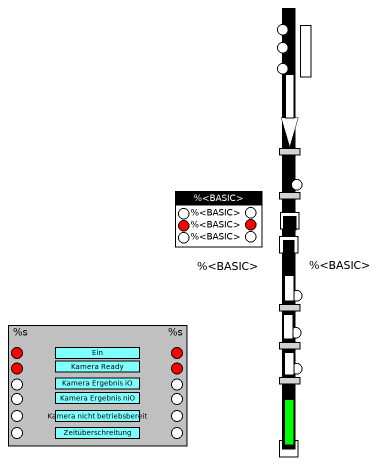
[picture p229: ZUFUEHRUNG_160POL (HMI screen)]
ellipse at (269,34)-(280,45): alarm colour if ST03_421_B63_5.BitInToCheck; tooltip ST03_421_B63_5
embedded screen at (273,66)-(290,139): SIGNS_ARROWDOWN
rounded rectangle at (272,204)-(291,221): alarm colour if ST03_422_B64_0.BitInToCheck; tooltip ST03_422_B64_0
ellipse at (269,55)-(280,66): alarm colour if ST03_421_B63_6.BitInToCheck; tooltip ST03_421_B63_6
ellipse at (269,16)-(280,27): alarm colour if ST03_421_B63_4.BitInToCheck; tooltip ST03_421_B63_4
ellipse at (283,282)-(294,293): alarm colour if ST03_422_B64_3.BitInToCheck; tooltip ST03_422_B64_3
rounded rectangle at (271,432)-(290,449): alarm colour if ST03_422_B64_4.BitInToCheck; tooltip ST03_422_B64_4
embedded screen at (0,317)-(179,437): ZLIB_SENSOPART_2
rectangle at (276,266)-(286,291): invisible if ST03_160pol_Zufuehrung.CamResult < 11; alarm colour if ST03_160pol_Zufuehrung.CamResult = 99
rectangle at (276,267)-(286,293): invisible if ST03_160pol_Zufuehrung.CamResult >= 11 OR NOT ST03_422_B64_3.BitInToCheck
rectangle at (276,391)-(286,437): invisible if NOT ST03_422_B64_4.BitInToCheck; alarm colour if ST03_Main.Result=RESULT_NOK
rectangle at (271,296)-(292,303): alarm colour if ST03_422_B64_1.ValveSensor; tooltip ST03_422_B64_1
rectangle at (271,184)-(292,191): alarm colour if ST03_421_B63_2.ValveSensor; tooltip ST03_421_B63_2
rectangle at (271,140)-(292,147): alarm colour if ST03_421_B63_0.ValveSensor; tooltip ST03_421_B63_0
rectangle at (275,212)-(286,226): alarm colour if ST03_421_B63_7.BitInToCheck
ellipse at (283,171)-(294,182): alarm colour if ST03_421_B63_7.BitInToCheck; tooltip ST03_421_B63_7
rounded rectangle at (292,17)-(303,69): alarm colour if ST03_Init_Lockings.b_freiFuerSG; tooltip b_freiFuerSG
embedded screen at (0,317)-(179,438): ZLIB_SENSOPART_6
ellipse at (282,319)-(293,330): alarm colour if ST03_423_B65_2.BitInToCheck; tooltip ST03_423_B65_2
rectangle at (275,305)-(285,330): invisible if ST03_160pol_Zufuehrung.CamResult2 < 11; alarm colour if ST03_160pol_Zufuehrung.CamResult2 = 99
rectangle at (275,306)-(285,331): invisible if ST03_160pol_Zufuehrung.CamResult2 >= 11 OR NOT ST03_423_B65_2.BitInToCheck
rectangle at (271,334)-(292,341): alarm colour if ST03_423_B65_0.ValveSensor; tooltip ST03_423_B65_0
ellipse at (283,355)-(294,366): alarm colour if ST03_423_B65_5.BitInToCheck; tooltip ST03_423_B65_5
rectangle at (276,343)-(286,365): invisible if ST03_160pol_Zufuehrung.CamResult3 < 11; alarm colour if ST03_160pol_Zufuehrung.CamResult3 = 99
rectangle at (276,344)-(286,367): invisible if ST03_160pol_Zufuehrung.CamResult3 >= 11 OR NOT ST03_423_B65_5.BitInToCheck
rectangle at (271,369)-(292,376): alarm colour if ST03_423_B65_4.ValveSensor; tooltip ST03_423_B65_4
rectangle at (299,245)-(374,270): text "%<BASIC>"; shows 'NIO Kamera'
rectangle at (187,246)-(265,271): text "%<BASIC>"; shows 'NIO Kamera'
rounded rectangle at (271,228)-(290,245): alarm colour if ST03_423_B66_0.BitInToCheck; tooltip ST03_423_B66_0
rectangle at (275,232)-(286,246): alarm colour if ST03_421_B63_7.BitInToCheck
rectangle at (167,196)-(254,239): shows 'Tank voll'
rectangle at (182,195)-(233,214): text "%<BASIC>"; shows 'bereit'
ellipse at (237,199)-(248,210): alarm colour if ST03_70U3_1.BitInToCheck
ellipse at (170,200)-(181,211): alarm colour if ST03_71U3_1.BitInToCheck
rectangle at (182,207)-(233,226): text "%<BASIC>"; shows 'Störung'
ellipse at (237,211)-(248,222): invisible if MP.ST03.SGM_3621; alarm colour if ST03_70U3_2.BitInToCheck
ellipse at (170,212)-(181,223): invisible if MP.ST03.SGM_3621; alarm colour if ST03_71U3_2.BitInToCheck
rectangle at (182,219)-(233,238): text "%<BASIC>"; shows 'Störung'
ellipse at (237,223)-(248,234): alarm colour if ST03_70U3_3.BitInToCheck
ellipse at (170,224)-(181,235): alarm colour if ST03_71U3_3.BitInToCheck
rectangle at (167,183)-(254,197): text "%<BASIC>"; shows 'li_Drucker_re'
3 more shapes without text or variables
6 elements of other kinds (tables, trends, ...) not read
*)

(* Visualisation zLibrary/ept/Zuführungen/ZUFUEHRUNG_191POL
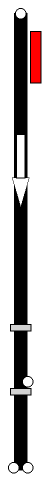
embedded screen at (9,126)-(26,199): SIGNS_ARROWDOWN
ellipse at (12,0)-(23,11): alarm colour if ST03_541_B69_0.BitInToCheck; tooltip ST03_541_B69_0
ellipse at (19,368)-(30,379): alarm colour if ST03_541_B69_6.BitInToCheck; tooltip ST03_541_B69_6
rectangle at (7,380)-(28,387): alarm colour if ST03_541_B69_4.ValveSensor; tooltip ST03_541_B69_3
rectangle at (7,316)-(28,323): alarm colour if ST03_541_B69_2.ValveSensor; tooltip ST03_541_B69_1
rounded rectangle at (27,23)-(38,75): alarm colour if ST03_Init_Lockings.b_freiFuerSG; tooltip b_freiFuerSG
ellipse at (19,454)-(30,465): alarm colour if ST03_542_B70_0.BitInToCheck; tooltip ST03_542_B70_0
ellipse at (5,454)-(16,465): alarm colour if ST03_541_B69_7.BitInToCheck; tooltip ST03_542_B70_0
2 more shapes without text or variables
*)

(* Visualisation zLibrary/ept/Zuführungen/ZUFUEHRUNG_206POL
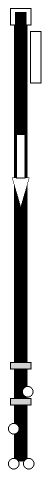
ellipse at (30,455)-(41,466): alarm colour if ST03_436_B68_1.BitInToCheck; tooltip ST03_436_B68_1
embedded screen at (19,131)-(36,204): SIGNS_ARROWDOWN
ellipse at (15,455)-(26,466): alarm colour if ST03_436_B68_2.BitInToCheck; tooltip ST03_436_B68_2
ellipse at (15,420)-(26,431): alarm colour if ST03_437_B68_4.BitInToCheck; tooltip ST03_437_B68_4
ellipse at (29,383)-(40,394): alarm colour if ST03_435_B67_7.BitInToCheck; tooltip ST03_435_B67_7
rectangle at (17,395)-(38,402): alarm colour if .ST03_435_B67_2.ValveSensor; tooltip .ST03_435_B67_2
rectangle at (17,359)-(38,366): alarm colour if ST03_435_B67_1.ValveSensor; tooltip ST03_435_B67_1
rounded rectangle at (17,5)-(38,22): alarm colour if ST03_435_B67_4.BitInToCheck; tooltip ST03_435_B67_4
rounded rectangle at (37,28)-(48,80): alarm colour if ST03_Init_Lockings.b_freiFuerSG; tooltip b_freiFuerSG
2 more shapes without text or variables
*)

(* Visualisation zLibrary/ept/Zuführungen/ZUFUEHRUNG_21POL
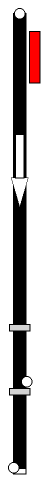
embedded screen at (9,126)-(26,199): SIGNS_ARROWDOWN
ellipse at (12,0)-(23,11): alarm colour if ST03_536_B69_0.BitInToCheck; tooltip ST03_536_B69_0
ellipse at (19,368)-(30,379): alarm colour if ST03_536_B69_6.BitInToCheck; tooltip ST03_536_B69_6
rectangle at (7,380)-(28,387): alarm colour if ST03_536_B69_4.ValveSensor; tooltip ST03_536_B69_3
rectangle at (7,316)-(28,323): alarm colour if ST03_536_B69_2.ValveSensor; tooltip ST03_536_B69_1
rounded rectangle at (27,23)-(38,75): alarm colour if ST03_Init_Lockings.b_freiFuerSG; tooltip b_freiFuerSG
rectangle at (11,460)-(24,466): alarm colour if ST03_537_B70_0.BitInToCheck; tooltip ST03_537_B70_0
ellipse at (6,454)-(17,465): alarm colour if ST03_536_B69_7.BitInToCheck; tooltip ST03_536_B69_7
2 more shapes without text or variables
*)

(* Visualisation zLibrary/ept/Zuführungen/ZUFUEHRUNG_268POL_102POL_NEU
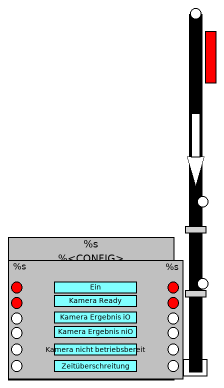
embedded screen at (179,202)-(196,275): SIGNS_ARROWDOWN
ellipse at (182,97)-(193,108): alarm colour if ST03_556_B69_0.BitInToCheck; tooltip ST03_556_B69_0
ellipse at (189,367)-(200,378): alarm colour if ST03_556_B69_6.BitInToCheck; tooltip ST03_556_B69_6
rectangle at (177,379)-(198,386): alarm colour if ST03_556_B69_4.ValveSensor; tooltip ST03_541_B69_3
rectangle at (177,315)-(198,322): alarm colour if ST03_556_B69_2.ValveSensor; tooltip ST03_541_B69_1
rounded rectangle at (175,448)-(199,465): alarm colour if ST03_556_B69_7.BitInToCheck; tooltip ST03_556_B69_7
rounded rectangle at (197,120)-(208,172): alarm colour if ST03_Init_Lockings.b_freiFuerSG; tooltip b_freiFuerSG
ellipse at (189,285)-(200,296): alarm colour if ST03_556_B69_5.BitInToCheck; tooltip ST03_556_B69_5
embedded screen at (0,326)-(166,469): ZLIB_SENSOPART_5
embedded screen at (0,349)-(175,468): ZLIB_SENSOPART_6
2 more shapes without text or variables
*)

(* Visualisation zLibrary/ept/Zuführungen/ZUFUEHRUNG_268POL_RP
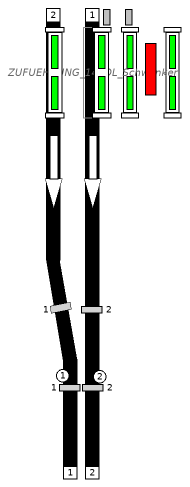
embedded screen at (73,127)-(90,200): SIGNS_ARROWDOWN
rounded rectangle at (74,0)-(88,14): text "1"; alarm colour if ST03_562_B69_0.BitInToCheck; tooltip ST03_562_B69_0
rounded rectangle at (74,458)-(88,471): text "2"; alarm colour if ST03_563_B70_7.BitInToCheck; tooltip ST03_563_B70_7
ellipse at (82,362)-(95,375): text "2"; alarm colour if ST03_563_B70_6.BitInToCheck; tooltip ST03_563_B70_6
rectangle at (71,376)-(92,383): alarm colour if ST03_563_B70_4.ValveSensor; tooltip ST03_563_B70_3
rectangle at (36,373)-(49,386): text "1"
rectangle at (92,373)-(105,386): text "2"
embedded screen at (110,19)-(170,110): ZUFUEHRUNG_268POL_RP_SCHWENKER
rectangle at (114,1)-(121,17): alarm colour if ST03_564_Y71_5.SensorInitIn[1].SensorSignal; tooltip ST03_564_Y71_5.SensorInitIn[1].SensorSignal
rectangle at (92,1)-(99,17): alarm colour if ST03_564_Y71_5.SensorWorkIn[1].SensorSignal; tooltip ST03_564_Y71_5.SensorWorkIn[1].SensorSignal
embedded screen at (72,19)-(91,110): ZUFUEHRUNG_14POL_Schwenker
rectangle at (48,376)-(69,383): alarm colour if ST03_562_B69_4.ValveSensor; tooltip ST03_564_Y71_1
rounded rectangle at (52,458)-(66,471): text "1"; alarm colour if ST03_562_B67_7.BitInToCheck; tooltip ST03_562_B67_7
ellipse at (45,361)-(58,374): text "1"; alarm colour if ST03_562_B69_6.BitInToCheck; tooltip ST03_562_B69_6
embedded screen at (34,19)-(100,110): ZUFUEHRUNG_268POL_RP_SCHWENKER
embedded screen at (34,127)-(51,200): SIGNS_ARROWDOWN
rectangle at (70,298)-(91,305): alarm colour if ST03_563_B70_2.ValveSensor; tooltip ST03_564_Y71_2
rectangle at (28,295)-(41,308): text "1"
rectangle at (91,295)-(104,308): text "2"
polygon at (39,294)-(60,305): alarm colour if ST03_562_B69_2.ValveSensor
rounded rectangle at (134,35)-(145,87): alarm colour if ST03_Init_Lockings.b_freiFuerSG; tooltip b_freiFuerSG
rounded rectangle at (35,0)-(49,14): text "2"; alarm colour if ST03_563_B70_0.BitInToCheck; tooltip ST03_563_B70_0
5 more shapes without text or variables
*)

(* Visualisation zLibrary/ept/Zuführungen/ZUFUEHRUNG_268POL_RP_SCHWENKER
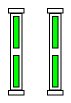
rectangle at (44,8)-(50,40): invisible if NOT $Reihe1$
rectangle at (44,47)-(50,79): invisible if NOT $Reihe1$
rounded rectangle at (39,0)-(55,5): invisible if NOT ST03_564_Y71_5.SensorWorkIn[1].SensorSignal; alarm colour if $Reihe1$; tooltip ST03_565_B72_0
rounded rectangle at (39,82)-(55,87): invisible if NOT ST03_564_Y71_5.SensorWorkIn[1].SensorSignal; alarm colour if $Reihe1$; tooltip ST03_565_B72_0
rectangle at (5,8)-(11,40): invisible if NOT $Reihe2$
rectangle at (5,47)-(11,79): invisible if NOT $Reihe2$
rounded rectangle at (0,0)-(16,5): invisible if NOT ST03_564_Y71_5.SensorWorkIn[1].SensorSignal; alarm colour if $Reihe2$; tooltip ST03_565_B72_1
rounded rectangle at (0,82)-(16,87): invisible if NOT ST03_564_Y71_5.SensorWorkIn[1].SensorSignal; alarm colour if $Reihe2$; tooltip ST03_565_B72_1
2 more shapes without text or variables
*)

(* Visualisation zLibrary/ept/Zuführungen/ZUFUEHRUNG_33POL
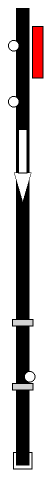
embedded screen at (9,126)-(26,199): SIGNS_ARROWDOWN
ellipse at (3,37)-(14,48): alarm colour if ST03_571_B69_0.BitInToCheck; tooltip ST03_501_B69_0
ellipse at (19,368)-(30,379): alarm colour if ST03_571_B69_6.BitInToCheck; tooltip ST03_501_B69_6
rectangle at (7,380)-(28,387): alarm colour if ST03_571_B69_5.ValveSensor; tooltip ST03_501_B69_3
rectangle at (7,316)-(28,323): alarm colour if ST03_571_B69_3.ValveSensor; tooltip ST03_501_B69_1
rounded rectangle at (8,449)-(27,466): alarm colour if ST03_571_B69_7.BitInToCheck; tooltip ST03_502_B70_0
rounded rectangle at (27,23)-(38,75): alarm colour if ST03_Init_Lockings.b_freiFuerSG; tooltip b_freiFuerSG
ellipse at (3,93)-(14,104): alarm colour if ST03_571_B69_1.BitInToCheck; tooltip ST03_501_B69_0
2 more shapes without text or variables
*)

(* Visualisation zLibrary/ept/Zuführungen/ZUFUEHRUNG_35POL
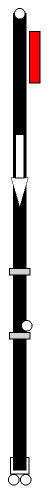
ellipse at (6,466)-(17,477): alarm colour if ST08_412_B58_6_35pol.BitInToCheck; tooltip ST08_412_B58_6_35pol
embedded screen at (9,126)-(26,199): SIGNS_ARROWDOWN
ellipse at (18,466)-(29,477): alarm colour if ST08_412_B58_5_35pol.BitInToCheck; tooltip ST08_412_B58_5_35pol
ellipse at (12,0)-(23,11): alarm colour if ST08_412_B58_4.BitInToCheck; tooltip ST08_412_B58_4
ellipse at (19,312)-(30,323): alarm colour if ST08_412_B58_7.BitInToCheck; tooltip ST08_412_B58_7
rectangle at (7,324)-(28,331): alarm colour if ST08_412_B58_2.ValveSensor; tooltip ST08_412_B58_2
rectangle at (7,260)-(28,267): alarm colour if ST08_412_B58_0.ValveSensor; tooltip ST08_412_B58_0
rounded rectangle at (8,449)-(27,466): alarm colour if ST08_412_B59_0.BitInToCheck; tooltip ST08_412_B59_0
rounded rectangle at (27,23)-(38,75): alarm colour if ST03_Init_Lockings.b_freiFuerSG; tooltip b_freiFuerSG
2 more shapes without text or variables
*)

(* Visualisation zLibrary/ept/Zuführungen/ZUFUEHRUNG_46POL
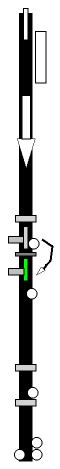
ellipse at (37,446)-(48,457): alarm colour if ST03_462_B70_1.BitInToCheck; tooltip ST03_462_B70_1
embedded screen at (23,92)-(41,165): SIGNS_ARROWDOWN
ellipse at (20,446)-(31,457): alarm colour if ST03_462_B70_2.BitInToCheck; tooltip ST03_462_B70_2
ellipse at (37,434)-(48,445): alarm colour if ST03_463_B70_7.BitInToCheck; tooltip ST03_463_B70_7
ellipse at (33,384)-(44,395): alarm colour if ST03_461_B69_7.BitInToCheck; tooltip ST03_461_B69_7
rectangle at (21,396)-(42,403): alarm colour if ST03_461_B69_2.ValveSensor; tooltip ST03_461_B69_2
rectangle at (21,361)-(42,368): alarm colour if ST03_461_B69_0.ValveSensor; tooltip ST03_461_B69_0
rounded rectangle at (41,28)-(52,80): alarm colour if ST03_Init_Lockings.b_freiFuerSG; tooltip b_freiFuerSG
rounded rectangle at (29,5)-(34,37): alarm colour if ST03_461_B69_4.BitInToCheck; tooltip ST03_461_B69_4
rectangle at (21,212)-(42,219): alarm colour if ST03_461_B69_5.ValveSensor; tooltip ST03_461_B69_5
rectangle at (14,233)-(30,240): invisible if NOT ST03_463_B70_5.ValveSensor; alarm colour if ST03_464_B71_6.BitInToCheck; tooltip ST03_464_B71_6; x offset ST03_CallFBs.ST03_463_B70_3_4_pos
rectangle at (29,223)-(34,246): invisible if NOT ST03_463_B70_5.ValveSensor; alarm colour if ST03_462_B70_0.BitInToCheck
rectangle at (29,255)-(34,278): invisible if NOT ST03_463_B70_6.ValveSensor
rectangle at (14,265)-(30,272): invisible if NOT ST03_463_B70_6.ValveSensor; alarm colour if ST03_464_B71_6.BitInToCheck; tooltip ST03_464_B71_6; x offset ST03_CallFBs.ST03_463_B70_3_4_pos
ellipse at (32,285)-(43,296): alarm colour if ST03_464_B71_7.BitInToCheck; tooltip ST03_464_B71_7
curve at (48,236)-(58,266): invisible if NOT ST03_463_B70_5.ValveSensor AND NOT NOT ST03_463_B70_5.ValveSensor
polygon at (42,264)-(51,272): invisible if NOT ST03_463_B70_5.ValveSensor AND NOT NOT ST03_463_B70_5.ValveSensor
ellipse at (34,235)-(45,246): alarm colour if ST03_462_B70_0.BitInToCheck; tooltip ST03_462_B70_0
2 more shapes without text or variables
*)

(* Visualisation zLibrary/ept/Zuführungen/ZUFUEHRUNG_48POL
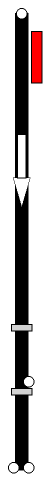
embedded screen at (9,126)-(26,199): SIGNS_ARROWDOWN
ellipse at (12,0)-(23,11): alarm colour if ST03_551_B69_0.BitInToCheck; tooltip ST03_541_B69_0
ellipse at (19,368)-(30,379): alarm colour if ST03_551_B69_6.BitInToCheck; tooltip ST03_541_B69_6
rectangle at (7,380)-(28,387): alarm colour if ST03_551_B69_4.ValveSensor; tooltip ST03_541_B69_3
rectangle at (7,316)-(28,323): alarm colour if ST03_551_B69_2.ValveSensor; tooltip ST03_541_B69_1
rounded rectangle at (27,23)-(38,75): alarm colour if ST03_Init_Lockings.b_freiFuerSG; tooltip b_freiFuerSG
ellipse at (4,454)-(15,465): alarm colour if ST03_552_B70_0.BitInToCheck; tooltip ST03_542_B70_0
ellipse at (19,454)-(30,465): alarm colour if ST03_551_B69_7.BitInToCheck; tooltip ST03_542_B70_0
2 more shapes without text or variables
*)

(* Visualisation zLibrary/ept/Zuführungen/ZUFUEHRUNG_72POL
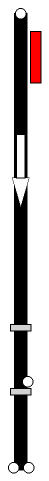
embedded screen at (9,126)-(26,199): SIGNS_ARROWDOWN
ellipse at (12,0)-(23,11): alarm colour if ST03_546_B69_0.BitInToCheck; tooltip ST03_541_B69_0
ellipse at (19,368)-(30,379): alarm colour if ST03_546_B69_6.BitInToCheck; tooltip ST03_541_B69_6
rectangle at (7,380)-(28,387): alarm colour if ST03_546_B69_4.ValveSensor; tooltip ST03_541_B69_3
rectangle at (7,316)-(28,323): alarm colour if ST03_546_B69_2.ValveSensor; tooltip ST03_541_B69_1
rounded rectangle at (27,23)-(38,75): alarm colour if ST03_Init_Lockings.b_freiFuerSG; tooltip b_freiFuerSG
ellipse at (5,454)-(16,465): alarm colour if ST03_547_B70_0.BitInToCheck; tooltip ST03_542_B70_0
ellipse at (20,454)-(31,465): alarm colour if ST03_546_B69_7.BitInToCheck; tooltip ST03_542_B70_0
2 more shapes without text or variables
*)

(* Visualisation zLibrary/ept/Zuführungen/ZUFUEHRUNG_74_91_168POL
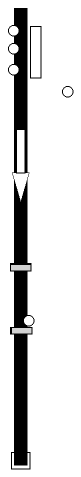
rounded rectangle at (8,444)-(27,461): invisible if NOT MP.ST03.SGM_3621; alarm colour if ST03_422_B64_4.BitInToCheck
ellipse at (5,35)-(16,46): invisible if MP.ST03.SGM_3621; alarm colour if ST08_412_B58_5.BitInToCheck
embedded screen at (9,121)-(26,194): SIGNS_ARROWDOWN
ellipse at (5,56)-(16,67): invisible if MP.ST03.SGM_3621 OR gTypeCode=379; alarm colour if ST08_412_B58_6.BitInToCheck
ellipse at (5,17)-(16,28): invisible if MP.ST03.SGM_3621; alarm colour if ST08_412_B58_4.BitInToCheck
ellipse at (19,307)-(30,318): invisible if MP.ST03.SGM_3621; alarm colour if ST08_412_B58_7.BitInToCheck
rectangle at (7,319)-(28,326): invisible if MP.ST03.SGM_3621; alarm colour if ST08_412_B58_2.ValveSensor
rectangle at (7,255)-(28,262): invisible if MP.ST03.SGM_3621; alarm colour if ST08_412_B58_0.ValveSensor
rounded rectangle at (8,444)-(27,461): invisible if MP.ST03.SGM_3621; alarm colour if ST08_412_B59_0.BitInToCheck; tooltip ST08_412_B59_0
rounded rectangle at (27,18)-(38,70): alarm colour if ST03_Init_Lockings.b_freiFuerSG; tooltip b_freiFuerSG
rectangle at (8,319)-(29,326): invisible if NOT MP.ST03.SGM_3621; alarm colour if ST03_421_B63_2.ValveSensor; tooltip ST03_421_B63_2
ellipse at (5,35)-(16,46): invisible if NOT MP.ST03.SGM_3621; alarm colour if ST03_421_B63_5.BitInToCheck; tooltip ST03_421_B63_5
ellipse at (59,78)-(70,89): invisible if NOT MP.ST03.SGM_3621; alarm colour if ST03_421_B63_6.BitInToCheck; tooltip ST03_421_B63_6
ellipse at (5,17)-(16,28): invisible if NOT MP.ST03.SGM_3621; alarm colour if ST03_421_B63_4.BitInToCheck; tooltip ST03_421_B63_4
rectangle at (7,256)-(28,263): invisible if NOT MP.ST03.SGM_3621; alarm colour if ST03_421_B63_0.ValveSensor; tooltip ST03_421_B63_0
ellipse at (20,307)-(31,318): invisible if NOT MP.ST03.SGM_3621; alarm colour if ST03_421_B63_7.BitInToCheck; tooltip ST03_421_B63_7
2 more shapes without text or variables
*)

(* Visualisation zLibrary/ept/Zuführungen/ZUFUEHRUNG_7POL
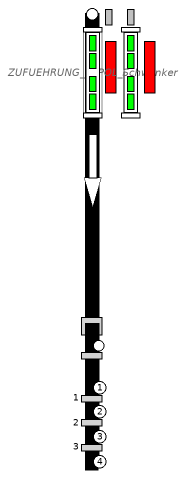
embedded screen at (16,126)-(33,199): SIGNS_ARROWDOWN
ellipse at (18,0)-(30,12): alarm colour if ST03_514_B71_7.BitInToCheck; tooltip ST03_514_B71_7
ellipse at (25,332)-(36,343): alarm colour if ST03_513_B70_4.BitInToCheck; tooltip ST03_513_B70_4
rectangle at (13,344)-(34,351): alarm colour if ST03_513_B70_3. ValveSensor; tooltip ST03_513_B70_3
rectangle at (13,309)-(34,327): alarm colour if ST03_513_B70_0.ValveSensor; tooltip ST03_513_B70_0
rounded rectangle at (37,33)-(48,85): alarm colour if ST03_Init_Lockings.b_freiFuerSG; tooltip b_freiFuerSG
ellipse at (25,447)-(38,460): text "4"; alarm colour if ST03_514_B71_6.BitInToCheck; tooltip ST03_514_B71_6
ellipse at (25,422)-(38,435): text "3"; alarm colour if ST03_514_B71_5.BitInToCheck; tooltip ST03_514_B71_5
rectangle at (13,436)-(34,443): alarm colour if ST03_514_B71_4.ValveSensor; tooltip ST03_514_B71_4
ellipse at (25,397)-(38,410): text "2"; alarm colour if ST03_514_B71_2.BitInToCheck; tooltip ST03_514_B71_2
rectangle at (13,411)-(34,418): alarm colour if ST03_514_B71_1.ValveSensor; tooltip ST03_514_B71_1
ellipse at (25,373)-(38,386): text "1"; alarm colour if ST03_513_B70_7.BitInToCheck; tooltip ST03_513_B70_7
rectangle at (13,387)-(34,394): alarm colour if ST03_513_B70_6.ValveSensor; tooltip ST03_513_B70_6
rectangle at (1,383)-(14,396): text "1"
rectangle at (1,408)-(14,421): text "2"
rectangle at (1,432)-(14,445): text "3"
embedded screen at (53,19)-(72,110): ZUFUEHRUNG_7POL_Schwenker
rectangle at (59,1)-(66,17): alarm colour if ST03_515_Y72_1.SensorInitIn[1].SensorSignal; tooltip ST03_515_Y72_1
rectangle at (37,1)-(44,17): alarm colour if ST03_515_Y72_1.SensorWorkIn[1].SensorSignal; tooltip ST03_515_Y72_1
embedded screen at (15,19)-(34,110): ZUFUEHRUNG_14POL_Schwenker
embedded screen at (15,19)-(34,110): ZUFUEHRUNG_7POL_Schwenker
rounded rectangle at (76,33)-(87,85): alarm colour if ST00_73_K4.BitInToCheck; tooltip ST00_73_K4
3 more shapes without text or variables
*)

(* Visualisation zLibrary/ept/Zuführungen/ZUFUEHRUNG_7POL_SCHWENKER
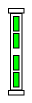
rectangle at (5,8)-(11,23): invisible if NOT ST03_512_XG1.BitInToCheck
rectangle at (5,25)-(11,40): invisible if NOT ST03_512_XG1.BitInToCheck
rectangle at (5,47)-(11,62): invisible if NOT ST03_512_XG1.BitInToCheck
rectangle at (5,64)-(11,79): invisible if NOT ST03_512_XG1.BitInToCheck
rounded rectangle at (0,0)-(16,5): invisible if ST03_515_Y72_1.SensorWorkIn[1].SensorSignal; alarm colour if ST03_512_XG1.BitInToCheck
rounded rectangle at (0,82)-(16,87): invisible if ST03_515_Y72_1.SensorWorkIn[1].SensorSignal; alarm colour if ST03_512_XG1.BitInToCheck
1 more shapes without text or variables
*)

(* Visualisation zLibrary/ept/Zuführungen/ZUFUEHRUNG_88POL
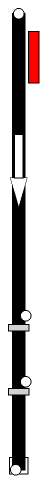
embedded screen at (9,126)-(26,199): SIGNS_ARROWDOWN
ellipse at (12,0)-(23,11): alarm colour if ST03_501_B69_0.BitInToCheck; tooltip ST03_501_B69_0
ellipse at (19,368)-(30,379): alarm colour if ST03_501_B69_6.BitInToCheck; tooltip ST03_501_B69_6
rectangle at (7,380)-(28,387): alarm colour if ST03_501_B69_3.ValveSensor; tooltip ST03_501_B69_3
rectangle at (7,316)-(28,323): alarm colour if ST03_501_B69_1.ValveSensor; tooltip ST03_501_B69_1
rounded rectangle at (8,449)-(27,466): alarm colour if ST03_502_B70_0.BitInToCheck; tooltip ST03_502_B70_0
rounded rectangle at (27,23)-(38,75): alarm colour if ST03_Init_Lockings.b_freiFuerSG; tooltip b_freiFuerSG
ellipse at (19,302)-(30,313): alarm colour if ST03_501_B69_5.BitInToCheck; tooltip ST03_501_B69_5
ellipse at (9,456)-(20,467): alarm colour if ST03_501_B69_7.BitInToCheck; tooltip ST03_501_B69_7
2 more shapes without text or variables
*)

(* Visualisation zLibrary/ept/Zuführungen/ZUFUEHRUNG_88POL_AMG
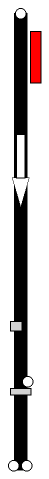
embedded screen at (9,126)-(26,199): SIGNS_ARROWDOWN
ellipse at (12,0)-(23,11): alarm colour if ST03_521_B69_0.BitInToCheck; tooltip ST03_521_B69_0
ellipse at (19,368)-(30,379): alarm colour if ST03_521_B69_6.BitInToCheck; tooltip ST03_521_B69_6
rectangle at (7,380)-(28,387): alarm colour if ST03_521_B69_4.ValveSensor; tooltip ST03_521_B69_3
rectangle at (7,313)-(19,323): alarm colour if ST03_521_B69_2.ValveSensor; tooltip ST03_521_B69_1
rounded rectangle at (27,23)-(38,75): alarm colour if ST03_Init_Lockings.b_freiFuerSG; tooltip b_freiFuerSG
ellipse at (5,452)-(16,463): alarm colour if ST03_521_B69_7.BitInToCheck; tooltip ST03_521_B69_7
ellipse at (18,452)-(29,463): alarm colour if ST03_522_B70_0.BitInToCheck; tooltip ST03_522_B70_0
2 more shapes without text or variables
*)

(* Visualisation zLibrary/ept/Zuführungen/ZUFUEHRUNG_92POL
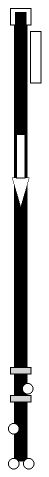
ellipse at (30,455)-(41,466): alarm colour if ST03_445_B70_1.BitInToCheck; tooltip ST03_445_B70_1
embedded screen at (19,131)-(36,204): SIGNS_ARROWDOWN
ellipse at (15,455)-(26,466): alarm colour if ST03_445_B70_2.BitInToCheck; tooltip ST03_445_B70_2
ellipse at (15,420)-(26,431): alarm colour if ST03_446_B70_4.BitInToCheck; tooltip ST03_446_B70_4
ellipse at (29,380)-(40,391): alarm colour if ST03_444_B69_7.BitInToCheck; tooltip ST03_444_B69_7
rectangle at (17,392)-(38,399): alarm colour if ST03_444_B69_2.ValveSensor; tooltip ST03_444_B69_2
rectangle at (17,364)-(38,371): alarm colour if ST03_444_B69_0.ValveSensor; tooltip ST03_444_B69_0
rounded rectangle at (17,5)-(38,22): alarm colour if ST03_435_B67_4.BitInToCheck; tooltip ST03_435_B67_4
rounded rectangle at (37,28)-(48,80): alarm colour if ST03_Init_Lockings.b_freiFuerSG; tooltip b_freiFuerSG
2 more shapes without text or variables
*)

(* Visualisation zLibrary/ept/Zuführungen/ZUFUEHRUNG_93POL
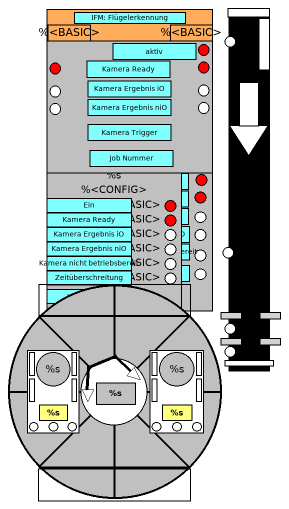
embedded screen at (40,160)-(206,303): ZLIB_SENSOPART_1
embedded screen at (40,160)-(175,303): ZLIB_SENSOPART_5
embedded screen at (0,276)-(215,493): ROUNDTABLE
embedded screen at (40,1)-(206,165): ZLIB_IFM
ellipse at (218,28)-(229,39): alarm colour if NOT ST02_FDB_40_B61.BitInToCheck; tooltip ST02_FDB_40_B61
embedded screen at (223,74)-(261,147): SIGNS_ARROWDOWN
ellipse at (218,315)-(229,326): alarm colour if ST00_72_X1_3.BitInToCheck; tooltip ST00_72_X1_3
rectangle at (214,304)-(235,311): alarm colour if ST00_74_Y2_5.SensorWorkIn[1].SensorSignal; tooltip ST00_74_Y2_5
rectangle at (253,304)-(274,311): alarm colour if ST00_74_Y2_5.SensorWorkIn[2].SensorSignal; tooltip ST00_74_Y2_5
rectangle at (214,330)-(235,337): alarm colour if NOT ST00_74_Y2_4.SensorWorkIn[1].SensorSignal; tooltip ST00_74_Y2_4
rectangle at (253,330)-(274,337): alarm colour if NOT ST00_74_Y2_4.SensorWorkIn[2].SensorSignal; tooltip ST00_74_Y2_4
rectangle at (222,342)-(263,363): invisible if gTypeCode<>4991
ellipse at (218,338)-(229,349): invisible if gTypeCode<>4991; alarm colour if ST02_FDB_80_B02.BitInToCheck; tooltip ST02_FDB_80_B02
rectangle at (218,352)-(267,358): invisible if gTypeCode<>4991
ellipse at (216,239)-(227,250): alarm colour if NOT ST02_FDB_40_B71.BitInToCheck; tooltip ST02_FDB_40_B71
rectangle at (225,149)-(259,156): alarm colour if ST02_FDB_54_B41.BitInToCheck
rounded rectangle at (252,10)-(263,62): alarm colour if ST03_Init_Lockings.b_freiFuerSG; tooltip b_freiFuerSG
rounded rectangle at (221,0)-(263,9): alarm colour if ST02_S1_40K01.BitInToCheck; tooltip ST02_S1_40K01
rectangle at (222,194)-(262,200): alarm colour if ST02_FDB_54_B21.ValveSensor
1 more shapes without text or variables
*)

(* Visualisation zLibrary/ept/Zuführungen/ZUFUEHRUNG_NOX_4POL
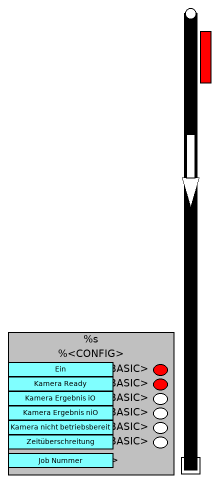
embedded screen at (174,126)-(191,199): SIGNS_ARROWDOWN
ellipse at (177,0)-(188,11): alarm colour if ST03_491_B69_0.BitInToCheck; tooltip ST03_491_B69_0
ellipse at (6,394)-(17,405): alarm colour if ST03_491_B69_5.BitInToCheck; tooltip ST03_491_B69_5
rectangle at (7,406)-(28,413): alarm colour if ST03_491_B69_2.ValveSensor; tooltip ST03_491_B69_2
rectangle at (7,371)-(28,378): alarm colour if ST03_491_B69_1.ValveSensor; tooltip ST03_491_B69_1
rounded rectangle at (173,449)-(192,466): alarm colour if ST03_491_B69_7.BitInToCheck; tooltip ST03_491_B69_7
rounded rectangle at (192,23)-(203,75): alarm colour if ST03_Init_Lockings.b_freiFuerSG; tooltip b_freiFuerSG
embedded screen at (0,324)-(166,467): ZLIB_SENSOPART_5
2 more shapes without text or variables
*)

(* Visualisation zLibrary/ept/Zuführungen/ZUFUEHRUNG_NOX_5_6POL
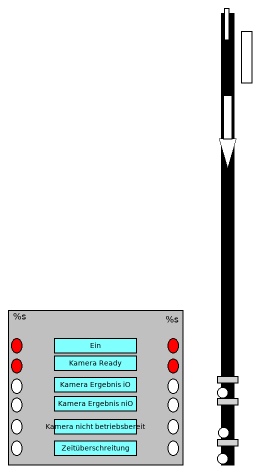
embedded screen at (274,87)-(291,160): SIGNS_ARROWDOWN
ellipse at (272,445)-(283,456): alarm colour if ST03_4x3_B70_1.BitInToCheck; tooltip ST03_4x3_B70_1
ellipse at (273,419)-(284,430): alarm colour if ST03_4x3_B70_0.BitInToCheck; tooltip ST03_4x3_B70_0
rectangle at (272,431)-(293,438): alarm colour if ST03_4x2_B69_7.ValveSensor; tooltip ST03_4x2_B69_7
rectangle at (272,390)-(293,397): alarm colour if ST03_4x2_B69_4.ValveSensor; tooltip ST03_4x2_B69_4
rounded rectangle at (296,23)-(307,75): alarm colour if ST03_Init_Lockings.b_freiFuerSG; tooltip b_freiFuerSG
rounded rectangle at (279,0)-(284,32): alarm colour if ST03_4x2_B69_0.BitInToCheck; tooltip ST03_4x2_B69_0
rounded rectangle at (272,368)-(293,375): alarm colour if ST03_4x2_B69_2.ValveSensor; tooltip ST03_4x2_B69_2
ellipse at (272,379)-(283,390): alarm colour if ST03_4x2_B69_5.BitInToCheck; tooltip ST03_4x2_B69_5
embedded screen at (63,302)-(238,457): ZLIB_SENSOPART_6
1 more shapes without text or variables
*)
